KUKA KRL data list: ps_ltc_geo_x1.dat

&ACCESS RVO2
&REL 17
&COMMENT Solda GUN X1 geometria
&PARAM DISKPATH = KRC:\R1\Program\SOLDA LTC
DEFDAT  ps_ltc_geo_x1
;FOLD EXTERNAL DECLARATIONS;%{PE}%MKUKATPBASIS,%CEXT,%VCOMMON,%P
;FOLD GRIPPERTECH EXT
EXT  H50 (INT  :IN,INT  :IN,INT  :IN,GRP_TYP  :IN )
;ENDFOLD (GRIPPERTECH EXT)
;FOLD SPOTTECH EXT
EXT  USERSPOT (S_COMMAND  :IN,SPOT_TYPE  :IN )
;ENDFOLD (SPOTTECH EXT)
;FOLD BASISTECH EXT;%{PE}%MKUKATPBASIS,%CEXT,%VEXT,%P
EXT  BAS (BAS_COMMAND  :IN,REAL  :IN )
DECL INT SUCCESS
;ENDFOLD (BASISTECH EXT)
;FOLD USER EXT;%{E}%MKUKATPUSER,%CEXT,%VEXT,%P
;Make your modifications here

;ENDFOLD (USER EXT)
;ENDFOLD (EXTERNAL DECLARATIONS)

;# ============ START PATH : swp_p13050r1_ltc_geo_x1 =============
DECL FDAT Fswp_60_0263={TOOL_NO 1,BASE_NO 2,IPO_FRAME #BASE,POINT2[] " "}
DECL SPOT_TYPE SS_OLP1={GUN 1,PAIR #FIRST,RETR #OPN,CLO_TM 0,PGNO1 1,PRESS1 1.0,PGNO2 0,PRESS2 0.0}
DECL E6POS Xswp_60_0263={X -275.645294,Y -980.43219,Z -166.443405,A 34.8704796,B 19.2542801,C 18.5798302,S 2,T 34,E1 -5647.1792,E2 0.0,E3 0.0,E4 0.0,E5 0.0,E6 0.0}
DECL FDAT Fswp_60_0267={TOOL_NO 1,BASE_NO 2,IPO_FRAME #BASE,POINT2[] " "}
DECL SPOT_TYPE SS_OLP2={GUN 1,PAIR #FIRST,RETR #OPN,CLO_TM 0,PGNO1 1,PRESS1 1.0,PGNO2 0,PRESS2 0.0}
DECL E6POS Xswp_60_0267={X -213.047607,Y -1048.96594,Z -164.542007,A 29.3044491,B 19.3898506,C 1.51828504,S 2,T 34,E1 -5647.19092,E2 0.0,E3 0.0,E4 0.0,E5 0.0,E6 0.0}
DECL FDAT Fswp_60_0283={TOOL_NO 1,BASE_NO 2,IPO_FRAME #BASE,POINT2[] " ",TQ_STATE FALSE}
DECL SPOT_TYPE SS_OLP3={GUN 1,PAIR #FIRST,RETR #OPN,CLO_TM 0,PGNO1 1,PRESS1 1.0,PGNO2 0,PRESS2 0.0}
DECL E6POS Xswp_60_0283={X 6.83988285,Y -1239.21399,Z 8.94310188,A 56.0263596,B 24.5332108,C -20.6315804,S 2,T 2,E1 -5181.69385,E2 0.0,E3 0.0,E4 0.0,E5 0.0,E6 0.0}
DECL SPOT_TYPE SS_OLP4={GUN 1,PAIR #FIRST,RETR #OPN,CLO_TM 0,PGNO1 1,PRESS1 1.0,PGNO2 0,PRESS2 0.0}
DECL SPOT_TYPE SS_OLP5={GUN 1,PAIR #FIRST,RETR #OPN,CLO_TM 0,PGNO1 1,PRESS1 1.0,PGNO2 0,PRESS2 0.0}
DECL FDAT Fswp_60_0349={TOOL_NO 1,BASE_NO 2,IPO_FRAME #BASE,POINT2[] " "}
DECL SPOT_TYPE SS_OLP6={GUN 1,PAIR #FIRST,RETR #OPN,CLO_TM 0,PGNO1 1,PRESS1 1.0,PGNO2 0,PRESS2 0.0}
DECL E6POS Xswp_60_0349={X 432.562195,Y -1705.31201,Z 116.379097,A 40.3507309,B 4.63222885,C -89.5844727,S 2,T 2,E1 -4540.75293,E2 0.0,E3 0.0,E4 0.0,E5 0.0,E6 0.0}
DECL FDAT Fswp_60_0355={TOOL_NO 1,BASE_NO 2,IPO_FRAME #BASE,POINT2[] " "}
DECL SPOT_TYPE SS_OLP7={GUN 1,PAIR #FIRST,RETR #OPN,CLO_TM 0,PGNO1 1,PRESS1 1.0,PGNO2 0,PRESS2 0.0}
DECL E6POS Xswp_60_0355={X 421.169403,Y -1718.13696,Z 279.697906,A 40.9335289,B -3.80524111,C -88.8869324,S 2,T 2,E1 -4540.78711,E2 0.0,E3 0.0,E4 0.0,E5 0.0,E6 0.0}
DECL FDAT Fswp_60_0317={TOOL_NO 1,BASE_NO 2,IPO_FRAME #BASE,POINT2[] " "}
DECL SPOT_TYPE SS_OLP8={GUN 1,PAIR #FIRST,RETR #OPN,CLO_TM 0,PGNO1 1,PRESS1 1.0,PGNO2 0,PRESS2 0.0}
DECL E6POS Xswp_60_0317={X 308.307007,Y -1610.21399,Z 6.46468401,A 127.521103,B -4.08989096,C 144.1259,S 2,T 10,E1 -4568.79297,E2 0.0,E3 0.0,E4 0.0,E5 0.0,E6 0.0}
DECL FDAT Fswp_60_0321={TOOL_NO 1,BASE_NO 2,IPO_FRAME #BASE,POINT2[] " ",TQ_STATE FALSE}
DECL SPOT_TYPE SS_OLP9={GUN 1,PAIR #FIRST,RETR #OPN,CLO_TM 0,PGNO1 1,PRESS1 1.0,PGNO2 0,PRESS2 0.0}
DECL E6POS Xswp_60_0321={X 337.849487,Y -1672.93506,Z -9.62210846,A 128.600006,B 1.93651104,C 143.567093,S 2,T 10,E1 -4568.6748,E2 0.0,E3 0.0,E4 0.0,E5 0.0,E6 0.0}
DECL FDAT Fswp_60_0325={TOOL_NO 1,BASE_NO 2,IPO_FRAME #BASE,POINT2[] " ",TQ_STATE FALSE}
DECL SPOT_TYPE SS_OLP10={GUN 1,PAIR #FIRST,RETR #OPN,CLO_TM 0,PGNO1 1,PRESS1 1.0,PGNO2 0,PRESS2 0.0}
DECL E6POS Xswp_60_0325={X 397.010406,Y -1691.29297,Z 3.9759531,A 119.003899,B -5.36455393,C 137.756195,S 2,T 10,E1 -4568.69678,E2 0.0,E3 0.0,E4 0.0,E5 0.0,E6 0.0}
DECL BASIS_SUGG_T LAST_BASIS={POINT1[] "PS01010001              ",POINT2[] "PS01010001              ",CP_PARAMS[] "CPDAT0                  ",PTP_PARAMS[] "PDAT0                   ",CONT[] "                        ",CP_VEL[] "2.0                     ",PTP_VEL[] " 100                    ",SPL_NAME[] "S0                      "}
DECL SPOT_SUGG_T LAST_SPOT={GUN[] "4                       ",RETR_CMD[] "#CLO                    ",CHOISE[] "#FIRST                  ",CLO_TM[] "1                       ",PGNO1[] "189                     ",PRESS1[] "0                       ",PGNO2[] "1                       ",PRESS2[] "0                       ",SPOT_PARAMS[] "NORMAL                  "}
DECL E6POS Xswp_60_0327={X -1825.44104,Y -6414.63623,Z 1659.75806,A -116.622902,B -6.43793201,C 136.093307,S 2,T 10,E1 -4568.69678,E2 0.0,E3 0.0,E4 0.0,E5 0.0,E6 0.0}
DECL FDAT Fswp_60_0327={TOOL_NO 1,BASE_NO 0,IPO_FRAME #BASE,POINT2[] " ",TQ_STATE FALSE}
DECL E6POS XP63={X 149.8685,Y -2567.51904,Z -128.437103,A 141.404694,B 27.8619308,C 99.6784897,S 2,T 10,E1 -4460.36279,E2 0.0,E3 0.0,E4 0.0,E5 0.0,E6 0.0}
DECL FDAT FP63={TOOL_NO 1,BASE_NO 2,IPO_FRAME #BASE,POINT2[] " ",TQ_STATE FALSE}
DECL PDAT PPDAT65={VEL 100.0,ACC 100.0,APO_DIST 100.0,APO_MODE #CDIS}
DECL E6POS XP112={X 128.800003,Y -2931.58496,Z -129.202301,A 55.0395699,B 45.2179985,C -42.0333595,S 2,T 2,E1 -3987.91797,E2 0.0,E3 0.0,E4 0.0,E5 0.0,E6 0.0}
DECL FDAT FP112={TOOL_NO 1,BASE_NO 2,IPO_FRAME #BASE,POINT2[] " ",TQ_STATE FALSE}
DECL PDAT PPDAT114={VEL 100.0,ACC 100.0,APO_DIST 100.0,APO_MODE #CDIS}
DECL PDAT PPDAT115={VEL 100.0,ACC 100.0,APO_DIST 100.0,APO_MODE #CDIS}
DECL E6POS XP113={X 223.016495,Y -1989.22095,Z 257.250488,A 40.7202988,B 3.102386,C -89.7601089,S 2,T 2,E1 -4540.78809,E2 0.0,E3 0.0,E4 0.0,E5 0.0,E6 0.0}
DECL FDAT FP113={TOOL_NO 1,BASE_NO 2,IPO_FRAME #BASE,POINT2[] " ",TQ_STATE FALSE}
DECL PDAT PPDAT116={VEL 100.0,ACC 100.0,APO_DIST 100.0,APO_MODE #CDIS}
DECL E6POS XP114={X 445.128204,Y -1749.01599,Z 250.443405,A 40.6904488,B -7.20178699,C -88.9869919,S 2,T 2,E1 -4540.78809,E2 0.0,E3 0.0,E4 0.0,E5 0.0,E6 0.0}
DECL FDAT FP114={TOOL_NO 1,BASE_NO 2,IPO_FRAME #BASE,POINT2[] " ",TQ_STATE FALSE}
DECL PDAT PP_OLP80={VEL 100.0,ACC 100.0,APO_DIST 0.0}
DECL PDAT PP_OLP81={VEL 100.0,ACC 100.0,APO_DIST 0.0}
DECL PDAT PPDAT117={VEL 100.0,ACC 100.0,APO_DIST 100.0,APO_MODE #CDIS}
DECL E6POS XP115={X 465.378387,Y -1730.63098,Z 102.938698,A 41.4731293,B 6.24935913,C -89.4617996,S 2,T 2,E1 -4540.75293,E2 0.0,E3 0.0,E4 0.0,E5 0.0,E6 0.0}
DECL FDAT FP115={TOOL_NO 1,BASE_NO 2,IPO_FRAME #BASE,POINT2[] " ",TQ_STATE FALSE}
DECL PDAT PP_OLP82={VEL 100.0,ACC 100.0,APO_DIST 100.0,APO_MODE #CDIS}
DECL E6POS Xlx695={X 247.467102,Y -1983.28699,Z 117.566002,A 40.3175316,B 0.397013813,C -89.5861206,S 2,T 2,E1 -4540.75293,E2 0.0,E3 0.0,E4 0.0,E5 0.0,E6 0.0}
DECL FDAT Flx695={TOOL_NO 1,BASE_NO 2,IPO_FRAME #BASE,POINT2[] " "}
DECL PDAT PPDAT119={VEL 100.0,ACC 100.0,APO_DIST 100.0,APO_MODE #CDIS}
DECL E6POS XP117={X -805.128296,Y -1482.06897,Z -24.73699,A 47.0636597,B 2.3741219,C -3.5756309,S 2,T 34,E1 -5647.1958,E2 0.0,E3 0.0,E4 0.0,E5 0.0,E6 0.0}
DECL FDAT FP117={TOOL_NO 1,BASE_NO 2,IPO_FRAME #BASE,POINT2[] " ",TQ_STATE FALSE}
DECL PDAT PPDAT120={VEL 100.0,ACC 100.0,APO_DIST 100.0,APO_MODE #CDIS}
DECL E6POS XP118={X -501.282806,Y -1183.51904,Z -151.957703,A 31.5826492,B 14.4653196,C -0.0970954373,S 2,T 34,E1 -5647.20117,E2 0.0,E3 0.0,E4 0.0,E5 0.0,E6 0.0}
DECL FDAT FP118={TOOL_NO 1,BASE_NO 2,IPO_FRAME #BASE,POINT2[] " ",TQ_STATE FALSE}
DECL PDAT PPDAT121={VEL 100.0,ACC 100.0,APO_DIST 100.0,APO_MODE #CDIS}
DECL PDAT PPDAT122={VEL 100.0,ACC 100.0,APO_DIST 100.0,APO_MODE #CDIS}
DECL E6POS XP120={X -240.307999,Y -1027.03699,Z -175.615204,A 32.5320892,B 19.41992,C 4.54465485,S 2,T 34,E1 -5647.1748,E2 0.0,E3 0.0,E4 0.0,E5 0.0,E6 0.0}
DECL FDAT FP120={TOOL_NO 1,BASE_NO 2,IPO_FRAME #BASE,POINT2[] " ",TQ_STATE FALSE}
DECL PDAT PPDAT123={VEL 100.0,ACC 100.0,APO_DIST 100.0,APO_MODE #CDIS}
DECL PDAT PP_OLP83={VEL 100.0,ACC 100.0,APO_DIST 100.0,APO_MODE #CDIS}
DECL E6POS Xlx696={X -459.795898,Y -1097.73706,Z -165.608002,A 36.6101303,B 19.1170197,C 8.19668961,S 2,T 34,E1 -5647.1748,E2 0.0,E3 0.0,E4 0.0,E5 0.0,E6 0.0}
DECL FDAT Flx696={TOOL_NO 1,BASE_NO 2,IPO_FRAME #BASE,POINT2[] " "}
DECL PDAT PP_OLP84={VEL 100.0,ACC 100.0,APO_DIST 100.0,APO_MODE #CDIS}
DECL E6POS Xlx697={X -805.127625,Y -1482.06995,Z -24.7408199,A 47.0636292,B 2.37426209,C -3.57572389,S 2,T 34,E1 -5647.1958,E2 0.0,E3 0.0,E4 0.0,E5 0.0,E6 0.0}
DECL FDAT Flx697={TOOL_NO 1,BASE_NO 2,IPO_FRAME #BASE,POINT2[] " "}
DECL PDAT PPDAT124={VEL 100.0,ACC 100.0,APO_DIST 80.0,APO_MODE #CDIS}
DECL E6POS XP122={X -339.747314,Y -1530.125,Z 57.2784996,A 62.6198311,B 11.3163099,C -12.12533,S 2,T 34,E1 -5181.66406,E2 0.0,E3 0.0,E4 0.0,E5 0.0,E6 0.0}
DECL FDAT FP122={TOOL_NO 1,BASE_NO 2,IPO_FRAME #BASE,POINT2[] " ",TQ_STATE FALSE}
DECL PDAT PPDAT125={VEL 100.0,ACC 50.0,APO_DIST 80.0,APO_MODE #CDIS}
DECL E6POS XP123={X -119.906601,Y -1419.73999,Z 23.3350296,A 66.8781586,B 12.7666798,C -15.6264,S 2,T 34,E1 -5181.68896,E2 0.0,E3 0.0,E4 0.0,E5 0.0,E6 0.0}
DECL FDAT FP123={TOOL_NO 1,BASE_NO 2,IPO_FRAME #BASE,POINT2[] " ",TQ_STATE FALSE}
DECL PDAT PPDAT126={VEL 100.0,ACC 50.0,APO_DIST 50.0,APO_MODE #CDIS}
DECL E6POS XP124={X -47.9475403,Y -1344.42505,Z 30.1196709,A 61.2519112,B 11.1653605,C -16.7942009,S 2,T 34,E1 -5181.68896,E2 0.0,E3 0.0,E4 0.0,E5 0.0,E6 0.0}
DECL FDAT FP124={TOOL_NO 1,BASE_NO 2,IPO_FRAME #BASE,POINT2[] " ",TQ_STATE FALSE}
DECL PDAT PPDAT127={VEL 100.0,ACC 50.0,APO_DIST 10.0,APO_MODE #CDIS}
DECL E6POS XP125={X -13.6633902,Y -1303.02698,Z 7.46283007,A 59.4785385,B 22.2280293,C -12.3178396,S 2,T 2,E1 -5181.68994,E2 0.0,E3 0.0,E4 0.0,E5 0.0,E6 0.0}
DECL FDAT FP125={TOOL_NO 1,BASE_NO 2,IPO_FRAME #BASE,POINT2[] " ",TQ_STATE FALSE}
DECL PDAT PP_OLP85={VEL 100.0,ACC 100.0,APO_DIST 0.0}
DECL PDAT PPDAT128={VEL 100.0,ACC 100.0,APO_DIST 15.0,APO_MODE #CDIS}
DECL E6POS XP126={X -48.0881805,Y -1344.44995,Z 26.9599705,A 59.0536118,B 21.2694607,C -19.8021393,S 2,T 2,E1 -5181.69092,E2 0.0,E3 0.0,E4 0.0,E5 0.0,E6 0.0}
DECL FDAT FP126={TOOL_NO 1,BASE_NO 2,IPO_FRAME #BASE,POINT2[] " ",TQ_STATE FALSE}
DECL PDAT PPDAT129={VEL 100.0,ACC 100.0,APO_DIST 20.0,APO_MODE #CDIS}
DECL E6POS XP127={X -141.712997,Y -1441.54504,Z 32.7751389,A 65.8396912,B 14.4452696,C -20.0396709,S 2,T 34,E1 -5181.68896,E2 0.0,E3 0.0,E4 0.0,E5 0.0,E6 0.0}
DECL FDAT FP127={TOOL_NO 1,BASE_NO 2,IPO_FRAME #BASE,POINT2[] " ",TQ_STATE FALSE}
DECL PDAT PPDAT134={VEL 100.0,ACC 100.0,APO_DIST 30.0,APO_MODE #CDIS}
DECL E6POS XP132={X -103.123703,Y -1698.18103,Z 59.301899,A 62.4764595,B 22.6058006,C -7.61601782,S 2,T 2,E1 -5181.7041,E2 0.0,E3 0.0,E4 0.0,E5 0.0,E6 0.0}
DECL FDAT FP132={TOOL_NO 1,BASE_NO 2,IPO_FRAME #BASE,POINT2[] " ",TQ_STATE FALSE}
DECL E6POS XP134={X 375.866486,Y -2553.52197,Z 94.818222,A 62.3175812,B 37.8605804,C -34.3857384,S 2,T 2,E1 -4175.70215,E2 0.0,E3 0.0,E4 0.0,E5 0.0,E6 0.0}
DECL FDAT FP134={TOOL_NO 1,BASE_NO 2,IPO_FRAME #BASE,POINT2[] " ",TQ_STATE FALSE}
DECL PDAT PPDAT136={VEL 100.0,ACC 100.0,APO_DIST 50.0,APO_MODE #CDIS}
DECL E6POS XP135={X 219.481094,Y -2785.84912,Z -130.159302,A 126.799698,B 53.5773201,C 39.0210495,S 2,T 10,E1 -4184.32813,E2 0.0,E3 0.0,E4 0.0,E5 0.0,E6 0.0}
DECL FDAT FP135={TOOL_NO 1,BASE_NO 2,IPO_FRAME #BASE,POINT2[] " ",TQ_STATE FALSE}
DECL PDAT PPDAT137={VEL 100.0,ACC 100.0,APO_DIST 100.0,APO_MODE #CDIS}
DECL PDAT PPDAT138={VEL 100.0,ACC 100.0,APO_DIST 100.0,APO_MODE #CDIS}
DECL E6POS XP136={X 429.565491,Y -1841.61304,Z -4.86375713,A 129.667999,B -2.37908912,C 148.920502,S 2,T 10,E1 -4568.75293,E2 0.0,E3 0.0,E4 0.0,E5 0.0,E6 0.0}
DECL FDAT FP136={TOOL_NO 1,BASE_NO 2,IPO_FRAME #BASE,POINT2[] " ",TQ_STATE FALSE}
DECL PDAT PP_OLP88={VEL 100.0,ACC 100.0,APO_DIST 100.0,APO_MODE #CDIS}
DECL E6POS Xlx698={X 292.525299,Y -1643.73096,Z -4.86532784,A 129.667999,B -2.37911105,C 148.920502,S 2,T 10,E1 -4568.75293,E2 0.0,E3 0.0,E4 0.0,E5 0.0,E6 0.0}
DECL FDAT Flx698={TOOL_NO 1,BASE_NO 2,IPO_FRAME #BASE,POINT2[] " "}
DECL PDAT PP_OLP89={VEL 100.0,ACC 100.0,APO_DIST 0.0}
DECL PDAT PPDAT139={VEL 100.0,ACC 100.0,APO_DIST 100.0,APO_MODE #CDIS}
DECL PDAT PPDAT140={VEL 100.0,ACC 100.0,APO_DIST 100.0,APO_MODE #CDIS}
DECL PDAT PPDAT141={VEL 100.0,ACC 100.0,APO_DIST 100.0,APO_MODE #CDIS}
DECL PDAT PPDAT146={VEL 100.0,ACC 100.0,APO_DIST 100.0,APO_MODE #CDIS}
DECL E6POS XP140={X 501.628906,Y -1918.77502,Z -26.8826199,A 116.119301,B 3.38413692,C 148.564102,S 2,T 10,E1 -4460.36279,E2 0.0,E3 0.0,E4 0.0,E5 0.0,E6 0.0}
DECL FDAT FP140={TOOL_NO 1,BASE_NO 2,IPO_FRAME #BASE,POINT2[] " ",TQ_STATE FALSE}
DECL PDAT PPDAT147={VEL 100.0,ACC 100.0,APO_DIST 100.0,APO_MODE #CDIS}
DECL E6POS XP141={X 149.8685,Y -2567.51904,Z -128.437103,A 141.404694,B 27.8619308,C 99.6784897,S 2,T 10,E1 -4460.36279,E2 0.0,E3 0.0,E4 0.0,E5 0.0,E6 0.0}
DECL FDAT FP141={TOOL_NO 1,BASE_NO 2,IPO_FRAME #BASE,POINT2[] " ",TQ_STATE FALSE}
DECL PDAT PP_OLP90={VEL 100.0,ACC 100.0,APO_DIST 100.0,APO_MODE #CDIS}
DECL E6POS Xlx610={X 192.240097,Y -2890.06006,Z -302.896515,A 132.393799,B 56.4223709,C 43.6062698,S 2,T 10,E1 -4184.32715,E2 0.0,E3 0.0,E4 0.0,E5 0.0,E6 0.0}
DECL FDAT Flx610={TOOL_NO 1,BASE_NO 2,IPO_FRAME #BASE,POINT2[] " "}
DECL PDAT PPDAT148={VEL 100.0,ACC 100.0,APO_DIST 100.0,APO_MODE #CDIS}
DECL E6POS XP142={X -20.6214809,Y -2868.67896,Z 427.8992,A 112.6278,B 26.7825699,C -22.8124199,S 2,T 2,E1 -3881.30811,E2 0.0,E3 0.0,E4 0.0,E5 0.0,E6 0.0}
DECL FDAT FP142={TOOL_NO 1,BASE_NO 2,IPO_FRAME #BASE,POINT2[] " ",TQ_STATE FALSE}
DECL PDAT PPDAT149={VEL 100.0,ACC 100.0,APO_DIST 100.0,APO_MODE #CDIS}
DECL E6POS XP143={X 301.243286,Y -1617.51001,Z 20.1037693,A 125.285301,B -8.34358597,C 149.555496,S 2,T 10,E1 -4568.78613,E2 0.0,E3 0.0,E4 0.0,E5 0.0,E6 0.0}
DECL FDAT FP143={TOOL_NO 1,BASE_NO 2,IPO_FRAME #BASE,POINT2[] " ",TQ_STATE FALSE}
DECL PDAT PPDAT150={VEL 100.0,ACC 100.0,APO_DIST 100.0,APO_MODE #CDIS}
DECL E6POS XP144={X 301.243286,Y -1617.51001,Z 20.1037693,A 125.285301,B -8.34358597,C 149.555496,S 2,T 10,E1 -4568.78613,E2 0.0,E3 0.0,E4 0.0,E5 0.0,E6 0.0}
DECL FDAT FP144={TOOL_NO 1,BASE_NO 2,IPO_FRAME #BASE,POINT2[] " ",TQ_STATE FALSE}
DECL PDAT PPDAT151={VEL 100.0,ACC 100.0,APO_DIST 100.0,APO_MODE #CDIS}
DECL E6POS Xswp_60_0315={X -1817.73596,Y -6538.56104,Z 1664.00903,A -105.512199,B -11.0989103,C 149.779205,S 2,T 10,E1 -4568.79785,E2 0.0,E3 0.0,E4 0.0,E5 0.0,E6 0.0}
DECL FDAT Fswp_60_0315={TOOL_NO 1,BASE_NO 0,IPO_FRAME #BASE,POINT2[] " ",TQ_STATE FALSE}
DECL E6POS XP145={X 291.662994,Y -1617.43896,Z -5.96740818,A 127.521301,B -4.09028482,C 144.125793,S 2,T 10,E1 -4568.79297,E2 0.0,E3 0.0,E4 0.0,E5 0.0,E6 0.0}
DECL FDAT FP145={TOOL_NO 1,BASE_NO 2,IPO_FRAME #BASE,POINT2[] " ",TQ_STATE FALSE}
DECL PDAT PPDAT152={VEL 100.0,ACC 100.0,APO_DIST 100.0,APO_MODE #CDIS}
DECL E6POS XP146={X 402.0242,Y -1685.71204,Z 23.6734409,A 111.884201,B -6.74503803,C 137.101501,S 2,T 10,E1 -4568.69678,E2 0.0,E3 0.0,E4 0.0,E5 0.0,E6 0.0}
DECL FDAT FP146={TOOL_NO 1,BASE_NO 2,IPO_FRAME #BASE,POINT2[] " ",TQ_STATE FALSE}
DECL PDAT PPDAT153={VEL 100.0,ACC 100.0,APO_DIST 100.0,APO_MODE #CDIS}
DECL E6POS XP147={X -11.8331299,Y -1323.75098,Z 0.671140611,A 58.5486107,B 17.0795193,C -15.2183399,S 2,T 34,E1 -5181.69092,E2 0.0,E3 0.0,E4 0.0,E5 0.0,E6 0.0}
DECL FDAT FP147={TOOL_NO 1,BASE_NO 2,IPO_FRAME #BASE,POINT2[] " ",TQ_STATE FALSE}
DECL PDAT PPDAT154={VEL 100.0,ACC 100.0,APO_DIST 80.0,APO_MODE #CDIS}
DECL PDAT PPDAT155={VEL 100.0,ACC 100.0,APO_DIST 100.0,APO_MODE #CDIS}
DECL E6POS Xswp_60_0331={X 319.516693,Y -1653.85706,Z -10.5840397,A 125.3731,B -3.16019797,C 145.238007,S 2,T 10,E1 -4568.69287,E2 0.0,E3 0.0,E4 0.0,E5 0.0,E6 0.0}
DECL FDAT Fswp_60_0331={TOOL_NO 1,BASE_NO 2,IPO_FRAME #BASE,POINT2[] " ",TQ_STATE FALSE}
DECL PDAT PPDAT156={VEL 100.0,ACC 100.0,APO_DIST 100.0,APO_MODE #CDIS}
DECL E6POS Xswp_60_0332={X 357.036591,Y -1691.21399,Z -9.36073685,A 128.599792,B 1.937621,C 143.567398,S 2,T 10,E1 -4568.6748,E2 0.0,E3 0.0,E4 0.0,E5 0.0,E6 0.0}
DECL FDAT Fswp_60_0332={TOOL_NO 1,BASE_NO 2,IPO_FRAME #BASE,POINT2[] " ",TQ_STATE FALSE}
DECL E6POS XP148={X 375.404388,Y -1714.22498,Z -8.3659811,A 128.599792,B 1.93763995,C 143.567505,S 2,T 10,E1 -4568.6748,E2 0.0,E3 0.0,E4 0.0,E5 0.0,E6 0.0}
DECL FDAT FP148={TOOL_NO 1,BASE_NO 2,IPO_FRAME #BASE,POINT2[] " ",TQ_STATE FALSE}
DECL PDAT PPDAT157={VEL 100.0,ACC 100.0,APO_DIST 80.0,APO_MODE #CDIS}
DECL E6POS XP149={X 387.077789,Y -1711.75806,Z 4.77827501,A 123.195396,B -3.82490492,C 140.115799,S 2,T 10,E1 -4568.68896,E2 0.0,E3 0.0,E4 0.0,E5 0.0,E6 0.0}
DECL FDAT FP149={TOOL_NO 1,BASE_NO 2,IPO_FRAME #BASE,POINT2[] " ",TQ_STATE FALSE}
DECL PDAT PPDAT158={VEL 100.0,ACC 100.0,APO_DIST 80.0,APO_MODE #CDIS}
DECL E6POS XP150={X 375.227386,Y -1691.30896,Z 21.6169395,A 116.706001,B -6.07782602,C 141.961105,S 2,T 10,E1 -4558.85889,E2 0.0,E3 0.0,E4 0.0,E5 0.0,E6 0.0}
DECL FDAT FP150={TOOL_NO 1,BASE_NO 2,IPO_FRAME #BASE,POINT2[] " ",TQ_STATE FALSE}
DECL PDAT PPDAT159={VEL 100.0,ACC 100.0,APO_DIST 100.0,APO_MODE #CDIS}
DECL E6POS XP151={X 355.217285,Y -1727.13794,Z 9.44879627,A 123.858902,B 0.442456514,C 146.9021,S 2,T 10,E1 -4533.8042,E2 0.0,E3 0.0,E4 0.0,E5 0.0,E6 0.0}
DECL FDAT FP151={TOOL_NO 1,BASE_NO 2,IPO_FRAME #BASE,POINT2[] " ",TQ_STATE FALSE}
DECL PDAT PPDAT160={VEL 100.0,ACC 100.0,APO_DIST 100.0,APO_MODE #CDIS}
DECL E6POS XP152={X 532.498291,Y -2000.23901,Z 8.68222904,A 118.759499,B 5.11184788,C 130.077805,S 2,T 10,E1 -4460.36279,E2 0.0,E3 0.0,E4 0.0,E5 0.0,E6 0.0}
DECL FDAT FP152={TOOL_NO 1,BASE_NO 2,IPO_FRAME #BASE,POINT2[] " ",TQ_STATE FALSE}
DECL PDAT PPDAT161={VEL 100.0,ACC 100.0,APO_DIST 100.0,APO_MODE #CDIS}
ENDDAT
